ABB RobotStudio station: Universo_EGM_1500_20220705-155238.rsstn

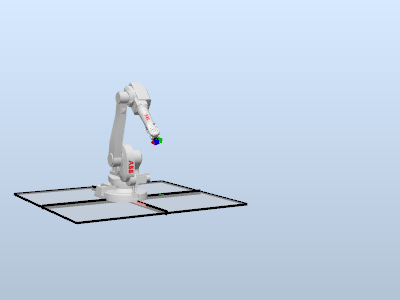
Station Universo_EGM_1500 (saved by RobotStudio 22.2.9947.0)
Controller IRB1600_6_145_1
  mechanical unit ROB_1: IRB1600_6_145__02, 6 joints, base frame (0, 0, 0) mm
Layout (positions relative to the parent item):
  - IRB1600_6_145__02 [mechanism, from Robots\IRB1600_6_145_G_02.rslib] at (0, 0, 0) mm; joint values [-0.0308, 0.2218, 0.4519, -1.1829, 0.1597, 0.9885] (rad or m)
